// TIA Portal V15.1 export
// export: Created 2024-06-21T08:41:02.8317921Z, ExportSetting WithDefaults, DisplayName Totally Integrated Automation Portal, DisplayVersion V15.1 Update 5, DisplayName TIA Portal Openness, DisplayVersion V15.1 Update 5, DisplayName SINAMICS Startdrive Advanced, DisplayVersion V15.1, DisplayName G130, G150, S120, S150, SINAMICS MV, S210, DisplayVersion V15.1, DisplayName G110M, G120, G120C, G120D, G120P, DisplayVersion V15.1, DisplayName STEP 7 Professional, DisplayVersion V15.1 Update 5, DisplayName STEP 7 Safety, DisplayVersion V15.1, DisplayName WinCC Professional, DisplayVersion V15.1 Update 5, DisplayName SIMATIC Visualization Architect, DisplayVersion V15.1
FUNCTION_BLOCK "LProcModeSelector"   // FB1708, FBD
TITLE = LModeSelector
{ S7_Optimized_Access := 'FALSE' }
AUTHOR : VCC
FAMILY : Control
NAME : ModeSel
VERSION : 1.0
// ================================================================================
// This module handles that only one mode is selected in the modezon, it also 
// handle interlocking between the HMIs. Each modezone can have 5 HMI.
// ================================================================================
// stored: AutoNumber false, IsIECCheckEnabled false, SetENOAutomatically False, UDAEnableTagReadback false
   VAR_INPUT
      I_StartPB { ExternalAccessible := 'False'; ExternalVisible := 'False'; ExternalWritable := 'False'} : Bool;   // Summary of Start buttons
      I_AlarmResetPB { ExternalAccessible := 'False'; ExternalVisible := 'False'; ExternalWritable := 'False'} : Bool;   // Summary of Alarm reset buttons
      I_SafetyNotOk { ExternalAccessible := 'False'; ExternalVisible := 'False'; ExternalWritable := 'False'} : Bool;   // Safety is not ok
      I_FailSafeResetAck { ExternalAccessible := 'False'; ExternalVisible := 'False'; ExternalWritable := 'False'} : Bool;   // F_Ack_Op FB in safety program is requesting value 9 on FailSafeReset output
      I_FailSafeAckID { ExternalAccessible := 'False'; ExternalVisible := 'False'; ExternalWritable := 'False'} : Int;   // F_Ack ID
      I_HMI1ForceMan { ExternalAccessible := 'False'; ExternalVisible := 'False'; ExternalWritable := 'False'} : Bool;   // Forced manual selected on HMI1
      I_HMI1SetPB { ExternalAccessible := 'False'; ExternalVisible := 'False'; ExternalWritable := 'False'} : Bool;   // Set PB activated on HMI1
      I_HMI1ResetPB { ExternalAccessible := 'False'; ExternalVisible := 'False'; ExternalWritable := 'False'} : Bool;   // Reset PB activated on HMI1
      I_HMI1StartPB { ExternalAccessible := 'False'; ExternalVisible := 'False'; ExternalWritable := 'False'} : Bool;   // Start PB activated on HMI1
      I_HMI1AlarmResetPB { ExternalAccessible := 'False'; ExternalVisible := 'False'; ExternalWritable := 'False'} : Bool;   // AlarmReset PB activated on HMI1
      I_HMI2ForceMan { ExternalAccessible := 'False'; ExternalVisible := 'False'; ExternalWritable := 'False'} : Bool;   // Forced manual selected on HMI2
      I_HMI2SetPB { ExternalAccessible := 'False'; ExternalVisible := 'False'; ExternalWritable := 'False'} : Bool;   // Set PB activated on HMI2
      I_HMI2ResetPB { ExternalAccessible := 'False'; ExternalVisible := 'False'; ExternalWritable := 'False'} : Bool;   // Reset PB activated on HMI2
      I_HMI2StartPB { ExternalAccessible := 'False'; ExternalVisible := 'False'; ExternalWritable := 'False'} : Bool;   // Start PB activated on HMI2
      I_HMI2AlarmResetPB { ExternalAccessible := 'False'; ExternalVisible := 'False'; ExternalWritable := 'False'} : Bool;   // AlarmReset PB activated on HMI2
      I_HMI3ForceMan { ExternalAccessible := 'False'; ExternalVisible := 'False'; ExternalWritable := 'False'} : Bool;   // Forced manual selected on HMI3
      I_HMI3SetPB { ExternalAccessible := 'False'; ExternalVisible := 'False'; ExternalWritable := 'False'} : Bool;   // Set PB activated on HMI3
      I_HMI3ResetPB { ExternalAccessible := 'False'; ExternalVisible := 'False'; ExternalWritable := 'False'} : Bool;   // Reset PB activated on HMI3
      I_HMI3StartPB { ExternalAccessible := 'False'; ExternalVisible := 'False'; ExternalWritable := 'False'} : Bool;   // Start PB activated on HMI
      I_HMI3AlarmResetPB { ExternalAccessible := 'False'; ExternalVisible := 'False'; ExternalWritable := 'False'} : Bool;   // AlarmReset PB activated on HMI3
      I_HMI4ForceMan { ExternalAccessible := 'False'; ExternalVisible := 'False'; ExternalWritable := 'False'} : Bool;   // Forced manual selected on HMI4
      I_HMI4SetPB { ExternalAccessible := 'False'; ExternalVisible := 'False'; ExternalWritable := 'False'} : Bool;   // Set PB activated on HMI4
      I_HMI4ResetPB { ExternalAccessible := 'False'; ExternalVisible := 'False'; ExternalWritable := 'False'} : Bool;   // Reset PB activated on HMI4
      I_HMI4StartPB { ExternalAccessible := 'False'; ExternalVisible := 'False'; ExternalWritable := 'False'} : Bool;   // Start PB activated on HMI4
      I_HMI4AlarmResetPB { ExternalAccessible := 'False'; ExternalVisible := 'False'; ExternalWritable := 'False'} : Bool;   // AlarmReset PB activated on HMI4
      I_HMI5ForceMan { ExternalAccessible := 'False'; ExternalVisible := 'False'; ExternalWritable := 'False'} : Bool;   // Forced manual selected on HMI5
      I_HMI5SetPB { ExternalAccessible := 'False'; ExternalVisible := 'False'; ExternalWritable := 'False'} : Bool;   // Set PB activated on HMI5
      I_HMI5ResetPB { ExternalAccessible := 'False'; ExternalVisible := 'False'; ExternalWritable := 'False'} : Bool;   // Reset PB activated on HMI5
      I_HMI5StartPB { ExternalAccessible := 'False'; ExternalVisible := 'False'; ExternalWritable := 'False'} : Bool;   // Start PB activated on HMI5
      I_HMI5AlarmResetPB { ExternalAccessible := 'False'; ExternalVisible := 'False'; ExternalWritable := 'False'} : Bool;   // AlarmReset PB activated on HMI5
   END_VAR
   VAR_OUTPUT
      O_PBSetPBResetAllAutoSel { ExternalAccessible := 'False'; ExternalVisible := 'False'; ExternalWritable := 'False'} : Struct   // Set PB activated - Reset PB activated - All HMI Auto selected
         HMI1SetPB { ExternalAccessible := 'False'; ExternalVisible := 'False'; ExternalWritable := 'False'} : Bool;   // Set PB activated on HMI1
         HMI1ResetPB { ExternalAccessible := 'False'; ExternalVisible := 'False'; ExternalWritable := 'False'} : Bool;   // Reset PB activated on HMI1
         HMI1AllHMIAutoSel { ExternalAccessible := 'False'; ExternalVisible := 'False'; ExternalWritable := 'False'} : Bool;   // All HMI Auto selected on HMI1
         HMI2SetPB { ExternalAccessible := 'False'; ExternalVisible := 'False'; ExternalWritable := 'False'} : Bool;   // Set PB activated on HMI2
         HMI2ResetPB { ExternalAccessible := 'False'; ExternalVisible := 'False'; ExternalWritable := 'False'} : Bool;   // Reset PB activated on HMI2
         HMI2AllHMIAutoSel { ExternalAccessible := 'False'; ExternalVisible := 'False'; ExternalWritable := 'False'} : Bool;   // All HMI Auto selected on HMI2
         HMI3SetPB { ExternalAccessible := 'False'; ExternalVisible := 'False'; ExternalWritable := 'False'} : Bool;   // Set PB activated on HMI3
         HMI3ResetPB { ExternalAccessible := 'False'; ExternalVisible := 'False'; ExternalWritable := 'False'} : Bool;   // Reset PB activated on HMI3
         HMI3AllHMIAutoSel { ExternalAccessible := 'False'; ExternalVisible := 'False'; ExternalWritable := 'False'} : Bool;   // All HMI Auto selected on HMI3
         HMI4SetPB { ExternalAccessible := 'False'; ExternalVisible := 'False'; ExternalWritable := 'False'} : Bool;   // Set PB activated on HMI4
         HMI4ResetPB { ExternalAccessible := 'False'; ExternalVisible := 'False'; ExternalWritable := 'False'} : Bool;   // Reset PB activated on HMI4
         HMI4AllHMIAutoSel { ExternalAccessible := 'False'; ExternalVisible := 'False'; ExternalWritable := 'False'} : Bool;   // All HMI Auto selected on HMI4
         HMI5SetPB { ExternalAccessible := 'False'; ExternalVisible := 'False'; ExternalWritable := 'False'} : Bool;   // Set PB activated on HMI5
         HMI5ResetPB { ExternalAccessible := 'False'; ExternalVisible := 'False'; ExternalWritable := 'False'} : Bool;   // Reset PB activated on HMI5
         HMI5AllHMIAutoSel { ExternalAccessible := 'False'; ExternalVisible := 'False'; ExternalWritable := 'False'} : Bool;   // All HMI Auto selected on HMI5
         StartPBSel { ExternalAccessible := 'False'; ExternalVisible := 'False'; ExternalWritable := 'False'} : Bool;   // Start is activated
         AlarmResetPBSel { ExternalAccessible := 'False'; ExternalVisible := 'False'; ExternalWritable := 'False'} : Bool;   // Alarm reset is activated
      END_STRUCT;
   END_VAR
   VAR_IN_OUT
      IO_FailsafeReset { ExternalAccessible := 'False'; ExternalVisible := 'False'; ExternalWritable := 'False'} : Int;   // Number to Failsafe to reset safety
   END_VAR
   VAR DB_SPECIFIC
      H_HMIHomeRunModeCmd : Word;   // Homerun Mode commands from HMI
      H_Anim : Word;   // Animation for HMI
      H_ActiveHMI : Int;   // Active HMI
      H_NameActiveHMI : String[25];   // Name of the Active HMI
      H_LockManTime : Int;   // Lock manual time
      H_HMI1ModeCmd : Word;   // Mode commands from HMI1
      H_HMI2ModeCmd : Word;   // Mode commands from HMI2
      H_HMI3ModeCmd : Word;   // Mode commands from HMI3
      H_HMI4ModeCmd : Word;   // Mode commands from HMI4
      H_HMI5ModeCmd : Word;   // Mode commands from HMI5. For operator panels, no S7_m_c
      HMI1AutoSel { ExternalAccessible := 'False'; ExternalVisible := 'False'; ExternalWritable := 'False'} : Bool;   // Auto selected on HMI1
      HMI1StepSel { ExternalAccessible := 'False'; ExternalVisible := 'False'; ExternalWritable := 'False'} : Bool;   // Step selected on HMI1
      HMI1HomeRunSel { ExternalAccessible := 'False'; ExternalVisible := 'False'; ExternalWritable := 'False'} : Bool;   // Homerun selected on HMI1
      HMI1ManualSel { ExternalAccessible := 'False'; ExternalVisible := 'False'; ExternalWritable := 'False'} : Bool;   // Manual selected on HMI1
      HMI1LockManual { ExternalAccessible := 'False'; ExternalVisible := 'False'; ExternalWritable := 'False'} : Bool;   // Lock manual for HMI1
      HMI1AllHMIAutoSel { ExternalAccessible := 'False'; ExternalVisible := 'False'; ExternalWritable := 'False'} : Bool;   // All HMI Auto selected on HMI1
      HMI1Start { ExternalAccessible := 'False'; ExternalVisible := 'False'; ExternalWritable := 'False'} : Bool;   // Start on HMI1
      HMI1AlarmReset { ExternalAccessible := 'False'; ExternalVisible := 'False'; ExternalWritable := 'False'} : Bool;   // AlarmReset on HMI1
      HMI1ResetTM { ExternalAccessible := 'False'; ExternalVisible := 'False'; ExternalWritable := 'False'} : Bool;   // Reset transport memory from HMI1
      HMI1ResetSeq { ExternalAccessible := 'False'; ExternalVisible := 'False'; ExternalWritable := 'False'} : Bool;   // Reset sequence from HMI1
      HMI1CycleFinished { ExternalAccessible := 'False'; ExternalVisible := 'False'; ExternalWritable := 'False'} : Bool;   // Cycle Finished from HMI1
      HMI1AlarmResetAck { ExternalAccessible := 'False'; ExternalVisible := 'False'; ExternalWritable := 'False'} : Bool;   // Alarm Reset acknowledge from HMI1
      HMI2AutoSel { ExternalAccessible := 'False'; ExternalVisible := 'False'; ExternalWritable := 'False'} : Bool;   // Auto selected on HMI2
      HMI2StepSel { ExternalAccessible := 'False'; ExternalVisible := 'False'; ExternalWritable := 'False'} : Bool;   // Step selected on HMI2
      HMI2HomeRunSel { ExternalAccessible := 'False'; ExternalVisible := 'False'; ExternalWritable := 'False'} : Bool;   // Homerun selected on HMI2
      HMI2ManualSel { ExternalAccessible := 'False'; ExternalVisible := 'False'; ExternalWritable := 'False'} : Bool;   // Manual selected on HMI2
      HMI2LockManual { ExternalAccessible := 'False'; ExternalVisible := 'False'; ExternalWritable := 'False'} : Bool;   // Lock manual for HMI2
      HMI2AllHMIAutoSel { ExternalAccessible := 'False'; ExternalVisible := 'False'; ExternalWritable := 'False'} : Bool;   // All HMI Auto selected on HMI2
      HMI2Start { ExternalAccessible := 'False'; ExternalVisible := 'False'; ExternalWritable := 'False'} : Bool;   // Start on HMI2
      HMI2AlarmReset { ExternalAccessible := 'False'; ExternalVisible := 'False'; ExternalWritable := 'False'} : Bool;   // AlarmReset on HMI2
      HMI2ResetTM { ExternalAccessible := 'False'; ExternalVisible := 'False'; ExternalWritable := 'False'} : Bool;   // Reset transport memory from HMI2
      HMI2ResetSeq { ExternalAccessible := 'False'; ExternalVisible := 'False'; ExternalWritable := 'False'} : Bool;   // Reset sequence from HMI2
      HMI2CycleFinished { ExternalAccessible := 'False'; ExternalVisible := 'False'; ExternalWritable := 'False'} : Bool;   // Cycle Finished from HMI2
      HMI2AlarmResetAck { ExternalAccessible := 'False'; ExternalVisible := 'False'; ExternalWritable := 'False'} : Bool;   // Alarm Reset acknowledge from HMI2
      HMI3AutoSel { ExternalAccessible := 'False'; ExternalVisible := 'False'; ExternalWritable := 'False'} : Bool;   // Auto selected on HMI3
      HMI3StepSel { ExternalAccessible := 'False'; ExternalVisible := 'False'; ExternalWritable := 'False'} : Bool;   // Step selected on HMI3
      HMI3HomeRunSel { ExternalAccessible := 'False'; ExternalVisible := 'False'; ExternalWritable := 'False'} : Bool;   // Homerun selected on HMI3
      HMI3ManualSel { ExternalAccessible := 'False'; ExternalVisible := 'False'; ExternalWritable := 'False'} : Bool;   // Manual selected on HMI3
      HMI3LockManual { ExternalAccessible := 'False'; ExternalVisible := 'False'; ExternalWritable := 'False'} : Bool;   // Lock manual for HMI3
      HMI3AllHMIAutoSel { ExternalAccessible := 'False'; ExternalVisible := 'False'; ExternalWritable := 'False'} : Bool;   // All HMI Auto selected on HMI3
      HMI3Start { ExternalAccessible := 'False'; ExternalVisible := 'False'; ExternalWritable := 'False'} : Bool;   // Start on HMI3
      HMI3AlarmReset { ExternalAccessible := 'False'; ExternalVisible := 'False'; ExternalWritable := 'False'} : Bool;   // AlarmReset on HMI3
      HMI3ResetTM { ExternalAccessible := 'False'; ExternalVisible := 'False'; ExternalWritable := 'False'} : Bool;   // Reset transport memory from HMI3
      HMI3ResetSeq { ExternalAccessible := 'False'; ExternalVisible := 'False'; ExternalWritable := 'False'} : Bool;   // Reset sequence from HMI3
      HMI3CycleFinished { ExternalAccessible := 'False'; ExternalVisible := 'False'; ExternalWritable := 'False'} : Bool;   // Cycle Finished from HMI3
      HMI3AlarmResetAck { ExternalAccessible := 'False'; ExternalVisible := 'False'; ExternalWritable := 'False'} : Bool;   // Alarm Reset acknowledge from 3
      HMI4AutoSel { ExternalAccessible := 'False'; ExternalVisible := 'False'; ExternalWritable := 'False'} : Bool;   // Auto selected on HMI4
      HMI4StepSel { ExternalAccessible := 'False'; ExternalVisible := 'False'; ExternalWritable := 'False'} : Bool;   // Step selected on HMI4
      HMI4HomeRunSel { ExternalAccessible := 'False'; ExternalVisible := 'False'; ExternalWritable := 'False'} : Bool;   // Homerun selected on HMI4
      HMI4ManualSel { ExternalAccessible := 'False'; ExternalVisible := 'False'; ExternalWritable := 'False'} : Bool;   // Manual selected on HMI4
      HMI4LockManual { ExternalAccessible := 'False'; ExternalVisible := 'False'; ExternalWritable := 'False'} : Bool;   // Lock manual for HMI4
      HMI4AllHMIAutoSel { ExternalAccessible := 'False'; ExternalVisible := 'False'; ExternalWritable := 'False'} : Bool;   // All HMI Auto selected on HMI4
      HMI4Start { ExternalAccessible := 'False'; ExternalVisible := 'False'; ExternalWritable := 'False'} : Bool;   // Start on HMI4
      HMI4AlarmReset { ExternalAccessible := 'False'; ExternalVisible := 'False'; ExternalWritable := 'False'} : Bool;   // AlarmReset on HMI4
      HMI4ResetTM { ExternalAccessible := 'False'; ExternalVisible := 'False'; ExternalWritable := 'False'} : Bool;   // Reset transport memory from HMI4
      HMI4ResetSeq { ExternalAccessible := 'False'; ExternalVisible := 'False'; ExternalWritable := 'False'} : Bool;   // Reset sequence from HMI4
      HMI4CycleFinished { ExternalAccessible := 'False'; ExternalVisible := 'False'; ExternalWritable := 'False'} : Bool;   // Cycle Finished from HMI4
      HMI4AlarmResetAck { ExternalAccessible := 'False'; ExternalVisible := 'False'; ExternalWritable := 'False'} : Bool;   // Alarm Reset acknowledge from HMI4
      HMI5AutoSel { ExternalAccessible := 'False'; ExternalVisible := 'False'; ExternalWritable := 'False'} : Bool;   // Auto selected on HMI5
      HMI5StepSel { ExternalAccessible := 'False'; ExternalVisible := 'False'; ExternalWritable := 'False'} : Bool;   // Step selected on HMI5
      HMI5HomeRunSel { ExternalAccessible := 'False'; ExternalVisible := 'False'; ExternalWritable := 'False'} : Bool;   // Homerun selected on HMI5
      HMI5ManualSel { ExternalAccessible := 'False'; ExternalVisible := 'False'; ExternalWritable := 'False'} : Bool;   // Manual selected on HMI5
      HMI5LockManual { ExternalAccessible := 'False'; ExternalVisible := 'False'; ExternalWritable := 'False'} : Bool;   // Lock manual for HMI5
      HMI5AllHMIAutoSel { ExternalAccessible := 'False'; ExternalVisible := 'False'; ExternalWritable := 'False'} : Bool;   // All HMI Auto selected on HMI5
      HMI5Start { ExternalAccessible := 'False'; ExternalVisible := 'False'; ExternalWritable := 'False'} : Bool;   // Start on HMI5
      HMI5AlarmReset { ExternalAccessible := 'False'; ExternalVisible := 'False'; ExternalWritable := 'False'} : Bool;   // AlarmReset on HMI5
      HMI5ResetTM { ExternalAccessible := 'False'; ExternalVisible := 'False'; ExternalWritable := 'False'} : Bool;   // Reset transport memory from HMI5
      HMI5ResetSeq { ExternalAccessible := 'False'; ExternalVisible := 'False'; ExternalWritable := 'False'} : Bool;   // Reset sequence from HMI5
      HMI5CycleFinished { ExternalAccessible := 'False'; ExternalVisible := 'False'; ExternalWritable := 'False'} : Bool;   // Cycle Finished from HMI5
      HMI5AlarmResetAck { ExternalAccessible := 'False'; ExternalVisible := 'False'; ExternalWritable := 'False'} : Bool;   // Alarm Reset acknowledge from HMI5
      HMIHomeRunRedo { ExternalAccessible := 'False'; ExternalVisible := 'False'; ExternalWritable := 'False'} : Bool;   // Redo after homerun from HMI
      HMIHomeRunWorkDone { ExternalAccessible := 'False'; ExternalVisible := 'False'; ExternalWritable := 'False'} : Bool;   // WorkDone after homerun from HMI
      LockManualTimeout { ExternalAccessible := 'False'; ExternalVisible := 'False'; ExternalWritable := 'False'} : Bool;   // Lock manual button timeout
      AllHmiAutoSel { ExternalAccessible := 'False'; ExternalVisible := 'False'; ExternalWritable := 'False'} : Bool;   // All Hmi Auto selected
      AlarmResetPBSel { ExternalAccessible := 'False'; ExternalVisible := 'False'; ExternalWritable := 'False'} : Bool;   // Alarm reset is activated
      AlarmResetPBSelReset { ExternalAccessible := 'False'; ExternalVisible := 'False'; ExternalWritable := 'False'} : Bool;   // Reset AlarmResetPBSel after predefined time
      AlarmResetPBSelResetPE { ExternalAccessible := 'False'; ExternalVisible := 'False'; ExternalWritable := 'False'} : Bool;   // Positive edge of AlarmResetPbSelReset
      FailSafeReset6Pulse { ExternalAccessible := 'False'; ExternalVisible := 'False'; ExternalWritable := 'False'} : Bool;   // Pulse to set value 6 on FailSafeReset Output
      FailSafeReset9Pulse { ExternalAccessible := 'False'; ExternalVisible := 'False'; ExternalWritable := 'False'} : Bool;   // Pulse to set value 9 on FailSafeReset Output
      ResetAlarmAckMemPulse { ExternalAccessible := 'False'; ExternalVisible := 'False'; ExternalWritable := 'False'} : Bool;   // Pulse to reset AlarmResetAckMem on negative edge of I_FailSafeResetAck
      AlarmResetAckMem { ExternalAccessible := 'False'; ExternalVisible := 'False'; ExternalWritable := 'False'} : Bool;   // memory : Pushbutton AlarmResetAck has been pushed on HMI
      StartPBSel { ExternalAccessible := 'False'; ExternalVisible := 'False'; ExternalWritable := 'False'} : Bool;   // Summary of the Start push buttons
      HMIStartPE { ExternalAccessible := 'False'; ExternalVisible := 'False'; ExternalWritable := 'False'} : Bool;   // Positive edge on start button from HMI
      HMIResetTMPE { ExternalAccessible := 'False'; ExternalVisible := 'False'; ExternalWritable := 'False'} : Bool;   // Positive edge on ResetTM button from HMI
      HMIResetSeqPE { ExternalAccessible := 'False'; ExternalVisible := 'False'; ExternalWritable := 'False'} : Bool;   // Positive edge on ResetSeq button from HMI
      HMIAlarmResetAckPE { ExternalAccessible := 'False'; ExternalVisible := 'False'; ExternalWritable := 'False'} : Bool;   // Positive edge on AlarmResetAck button from HMI
      HMILockManualPE { ExternalAccessible := 'False'; ExternalVisible := 'False'; ExternalWritable := 'False'} : Bool;   // Positive edge on LockManual button from HMI
      FailsafeReset { ExternalAccessible := 'False'; ExternalVisible := 'False'; ExternalWritable := 'False'} : Int;   // Number to Failsafe to reset safety
      ActiveHMI { ExternalAccessible := 'False'; ExternalVisible := 'False'; ExternalWritable := 'False'} : Int;   // Help memory for Active HMI
   END_VAR
   VAR
      TimerLockMan { ExternalAccessible := 'False'; ExternalVisible := 'False'; ExternalWritable := 'False'; S7_SetPoint := 'True'} : "LTimer";   // Timer on Lock manual
      TimerAlarmResetPB { ExternalAccessible := 'False'; ExternalVisible := 'False'; ExternalWritable := 'False'; S7_SetPoint := 'True'} : "LTimer";   // Timer on alarm reset
   END_VAR
   VAR_TEMP
      PHMI1AutoSel : Bool;   // Pulse Auto selected HMI1
      PHMI2AutoSel : Bool;   // Pulse Auto selected HMI2
      PHMI3AutoSel : Bool;   // Pulse Auto selected HMI3
      PHMI4AutoSel : Bool;   // Pulse Auto selected HMI4
      PHMI5AutoSel : Bool;   // Pulse Auto selected HMI5
   END_VAR
   VAR_TEMP   // added for the SCL form of the ladder/FBD networks
      _w1 : Bool;
      _w2 : Bool;
      _w3 : Bool;
      _w4 : Bool;
      _w5 : Bool;
   END_VAR
BEGIN

REGION Network 1: **** 1 - Inputs **** Extract the modeselection from HMI 1
   // Extract the modeselection from HMI 1
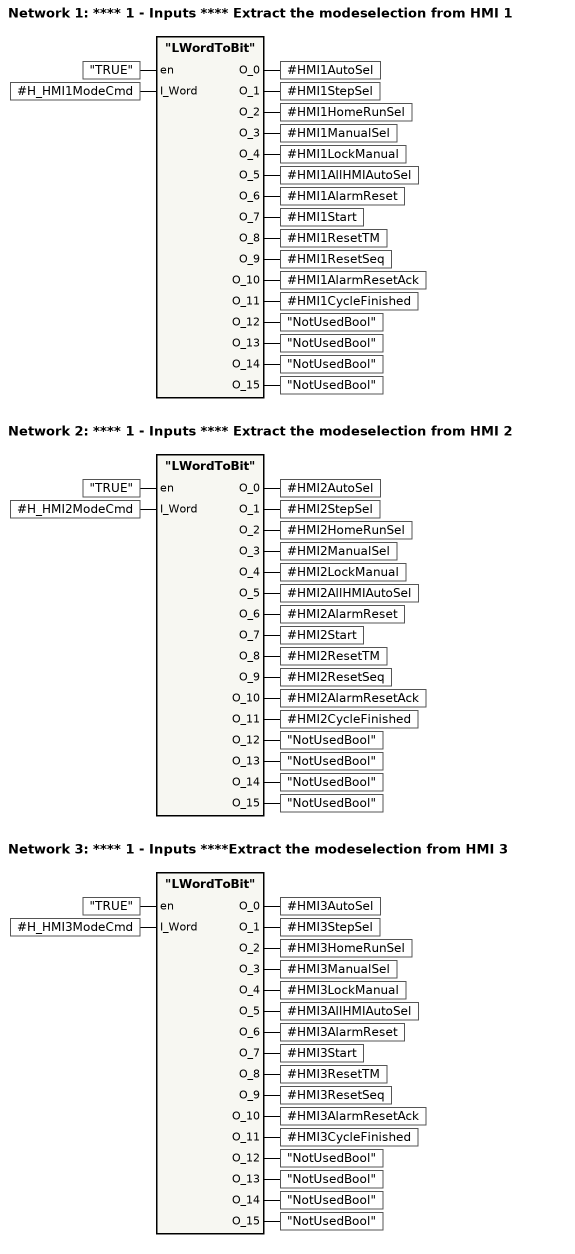
   IF "TRUE" THEN
       "LWordToBit"(I_Word := #H_HMI1ModeCmd,
                    O_0 => #HMI1AutoSel,
                    O_1 => #HMI1StepSel,
                    O_2 => #HMI1HomeRunSel,
                    O_3 => #HMI1ManualSel,
                    O_4 => #HMI1LockManual,
                    O_5 => #HMI1AllHMIAutoSel,
                    O_6 => #HMI1AlarmReset,
                    O_7 => #HMI1Start,
                    O_8 => #HMI1ResetTM,
                    O_9 => #HMI1ResetSeq,
                    O_10 => #HMI1AlarmResetAck,
                    O_11 => #HMI1CycleFinished,
                    O_12 => "NotUsedBool",
                    O_13 => "NotUsedBool",
                    O_14 => "NotUsedBool",
                    O_15 => "NotUsedBool");
   END_IF;
END_REGION

REGION Network 2: **** 1 - Inputs **** Extract the modeselection from HMI 2
   // Extract the modeselection from HMI 2
   IF "TRUE" THEN
       "LWordToBit"(I_Word := #H_HMI2ModeCmd,
                    O_0 => #HMI2AutoSel,
                    O_1 => #HMI2StepSel,
                    O_2 => #HMI2HomeRunSel,
                    O_3 => #HMI2ManualSel,
                    O_4 => #HMI2LockManual,
                    O_5 => #HMI2AllHMIAutoSel,
                    O_6 => #HMI2AlarmReset,
                    O_7 => #HMI2Start,
                    O_8 => #HMI2ResetTM,
                    O_9 => #HMI2ResetSeq,
                    O_10 => #HMI2AlarmResetAck,
                    O_11 => #HMI2CycleFinished,
                    O_12 => "NotUsedBool",
                    O_13 => "NotUsedBool",
                    O_14 => "NotUsedBool",
                    O_15 => "NotUsedBool");
   END_IF;
END_REGION

REGION Network 3: **** 1 - Inputs ****Extract the modeselection from HMI 3
   // Extract the modeselection from HMI 3
   IF "TRUE" THEN
       "LWordToBit"(I_Word := #H_HMI3ModeCmd,
                    O_0 => #HMI3AutoSel,
                    O_1 => #HMI3StepSel,
                    O_2 => #HMI3HomeRunSel,
                    O_3 => #HMI3ManualSel,
                    O_4 => #HMI3LockManual,
                    O_5 => #HMI3AllHMIAutoSel,
                    O_6 => #HMI3AlarmReset,
                    O_7 => #HMI3Start,
                    O_8 => #HMI3ResetTM,
                    O_9 => #HMI3ResetSeq,
                    O_10 => #HMI3AlarmResetAck,
                    O_11 => #HMI3CycleFinished,
                    O_12 => "NotUsedBool",
                    O_13 => "NotUsedBool",
                    O_14 => "NotUsedBool",
                    O_15 => "NotUsedBool");
   END_IF;
END_REGION

REGION Network 4: **** 1 - Inputs **** Extract the modeselection from HMI 4
   // Extract the modeselection from HMI 4
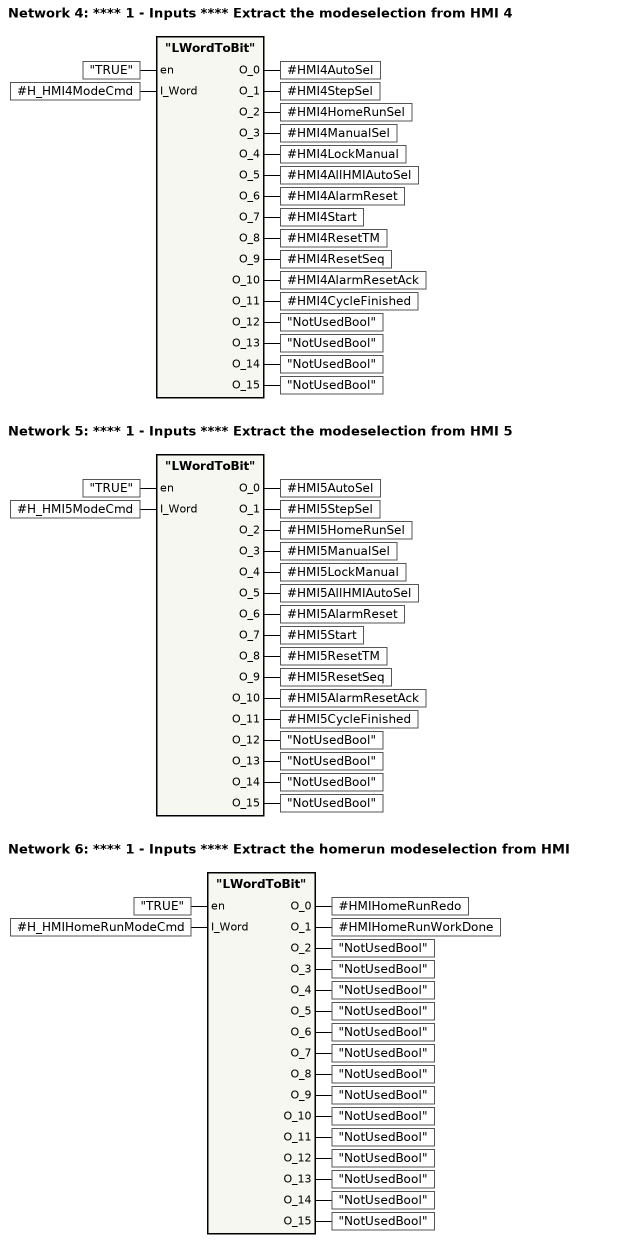
   IF "TRUE" THEN
       "LWordToBit"(I_Word := #H_HMI4ModeCmd,
                    O_0 => #HMI4AutoSel,
                    O_1 => #HMI4StepSel,
                    O_2 => #HMI4HomeRunSel,
                    O_3 => #HMI4ManualSel,
                    O_4 => #HMI4LockManual,
                    O_5 => #HMI4AllHMIAutoSel,
                    O_6 => #HMI4AlarmReset,
                    O_7 => #HMI4Start,
                    O_8 => #HMI4ResetTM,
                    O_9 => #HMI4ResetSeq,
                    O_10 => #HMI4AlarmResetAck,
                    O_11 => #HMI4CycleFinished,
                    O_12 => "NotUsedBool",
                    O_13 => "NotUsedBool",
                    O_14 => "NotUsedBool",
                    O_15 => "NotUsedBool");
   END_IF;
END_REGION

REGION Network 5: **** 1 - Inputs **** Extract the modeselection from HMI 5
   // Extract the modeselection from HMI 5
   IF "TRUE" THEN
       "LWordToBit"(I_Word := #H_HMI5ModeCmd,
                    O_0 => #HMI5AutoSel,
                    O_1 => #HMI5StepSel,
                    O_2 => #HMI5HomeRunSel,
                    O_3 => #HMI5ManualSel,
                    O_4 => #HMI5LockManual,
                    O_5 => #HMI5AllHMIAutoSel,
                    O_6 => #HMI5AlarmReset,
                    O_7 => #HMI5Start,
                    O_8 => #HMI5ResetTM,
                    O_9 => #HMI5ResetSeq,
                    O_10 => #HMI5AlarmResetAck,
                    O_11 => #HMI5CycleFinished,
                    O_12 => "NotUsedBool",
                    O_13 => "NotUsedBool",
                    O_14 => "NotUsedBool",
                    O_15 => "NotUsedBool");
   END_IF;
END_REGION

REGION Network 6: **** 1 - Inputs **** Extract the homerun modeselection from HMI
   // Extract the homerun modeselection from HMI
   IF "TRUE" THEN
       "LWordToBit"(I_Word := #H_HMIHomeRunModeCmd,
                    O_0 => #HMIHomeRunRedo,
                    O_1 => #HMIHomeRunWorkDone,
                    O_2 => "NotUsedBool",
                    O_3 => "NotUsedBool",
                    O_4 => "NotUsedBool",
                    O_5 => "NotUsedBool",
                    O_6 => "NotUsedBool",
                    O_7 => "NotUsedBool",
                    O_8 => "NotUsedBool",
                    O_9 => "NotUsedBool",
                    O_10 => "NotUsedBool",
                    O_11 => "NotUsedBool",
                    O_12 => "NotUsedBool",
                    O_13 => "NotUsedBool",
                    O_14 => "NotUsedBool",
                    O_15 => "NotUsedBool");
   END_IF;
END_REGION

REGION Network 7: **** 1 - Inputs **** All HMI Auto selected
   // All HMI Auto selected
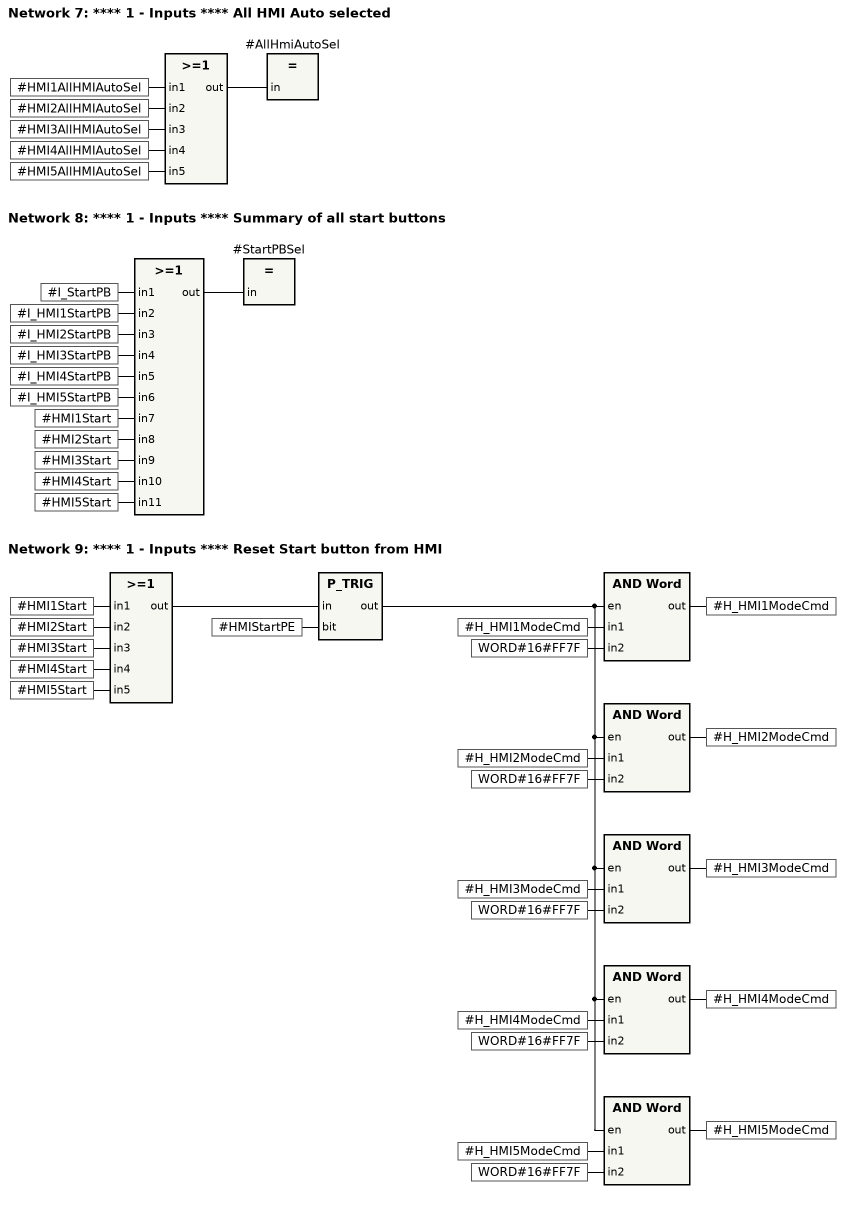
   #AllHmiAutoSel := #HMI1AllHMIAutoSel OR #HMI2AllHMIAutoSel OR #HMI3AllHMIAutoSel OR #HMI4AllHMIAutoSel OR #HMI5AllHMIAutoSel;
END_REGION

REGION Network 8: **** 1 - Inputs **** Summary of all start buttons
   // Summary of all start buttons
   #StartPBSel := #I_StartPB OR #I_HMI1StartPB OR #I_HMI2StartPB OR #I_HMI3StartPB OR #I_HMI4StartPB OR #I_HMI5StartPB OR #HMI1Start OR #HMI2Start OR #HMI3Start OR #HMI4Start OR #HMI5Start;
END_REGION

REGION Network 9: **** 1 - Inputs **** Reset Start button from HMI
   // Reset Start button from HMI
   #_w1 := #HMI1Start OR #HMI2Start OR #HMI3Start OR #HMI4Start OR #HMI5Start;
   #_w2 := #_w1 AND NOT #HMIStartPE;   // rising edge
   #HMIStartPE := #_w1;
   IF #_w2 THEN
       #H_HMI1ModeCmd := #H_HMI1ModeCmd AND WORD#16#FF7F;
       #H_HMI2ModeCmd := #H_HMI2ModeCmd AND WORD#16#FF7F;
       #H_HMI3ModeCmd := #H_HMI3ModeCmd AND WORD#16#FF7F;
       #H_HMI4ModeCmd := #H_HMI4ModeCmd AND WORD#16#FF7F;
       #H_HMI5ModeCmd := #H_HMI5ModeCmd AND WORD#16#FF7F;
   END_IF;
END_REGION

REGION Network 10: **** 1 - Inputs **** Summary of all alarm reset buttons
   // Summary of all alarm reset buttons
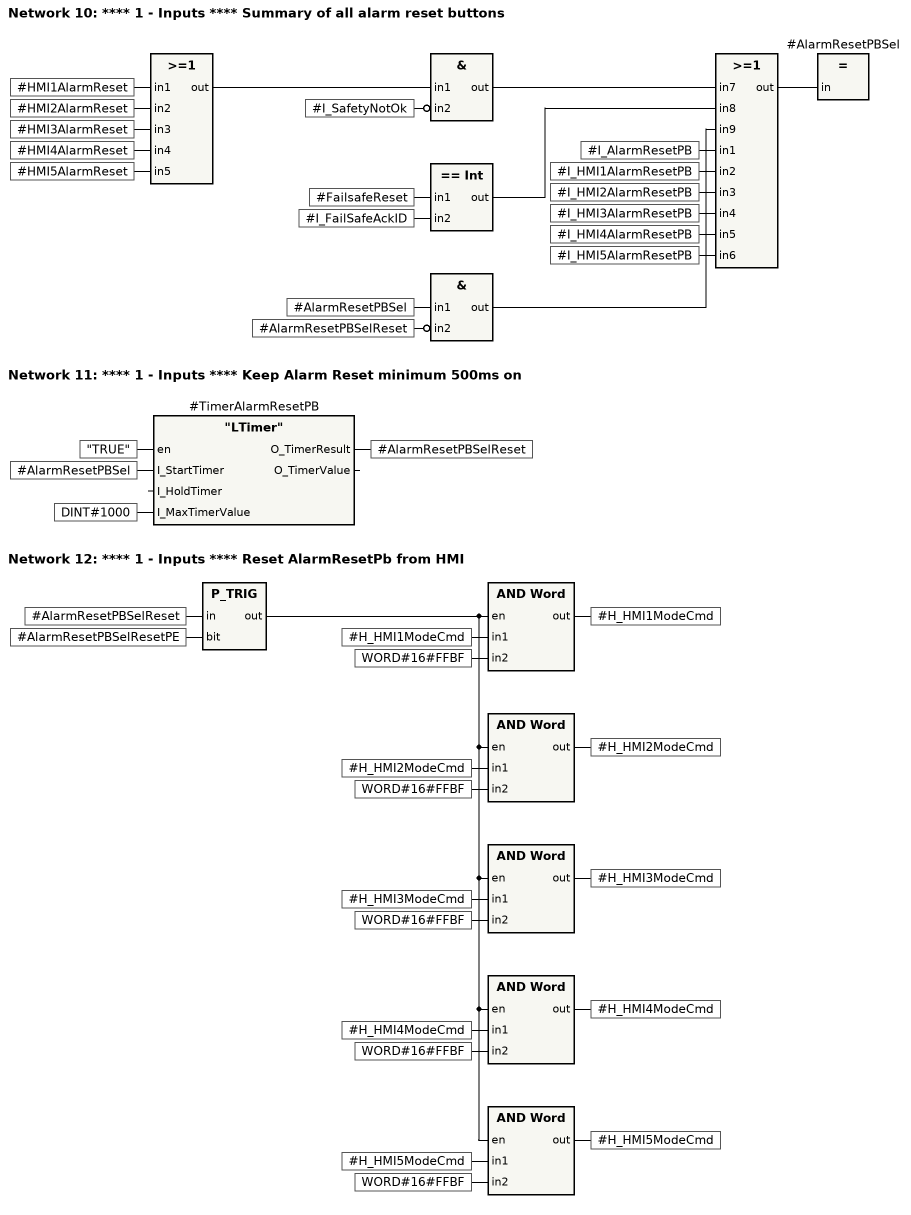
   #AlarmResetPBSel := ((#HMI1AlarmReset OR #HMI2AlarmReset OR #HMI3AlarmReset OR #HMI4AlarmReset OR #HMI5AlarmReset) AND NOT #I_SafetyNotOk) OR (#FailsafeReset = #I_FailSafeAckID) OR (#AlarmResetPBSel AND NOT #AlarmResetPBSelReset) OR #I_AlarmResetPB OR #I_HMI1AlarmResetPB OR #I_HMI2AlarmResetPB OR #I_HMI3AlarmResetPB OR #I_HMI4AlarmResetPB OR #I_HMI5AlarmResetPB;
END_REGION

REGION Network 11: **** 1 - Inputs **** Keep Alarm Reset minimum 500ms on
   // Keep Alarm Reset minimum 500ms on
   IF "TRUE" THEN
       #TimerAlarmResetPB(I_StartTimer := #AlarmResetPBSel,   // "LTimer"
                          I_MaxTimerValue := DINT#1000,
                          O_TimerResult => #AlarmResetPBSelReset);
   END_IF;
END_REGION

REGION Network 12: **** 1 - Inputs **** Reset AlarmResetPb from HMI
   // Reset AlarmResetPb from HMI
   #_w1 := #AlarmResetPBSelReset AND NOT #AlarmResetPBSelResetPE;   // rising edge
   #AlarmResetPBSelResetPE := #AlarmResetPBSelReset;
   IF #_w1 THEN
       #H_HMI1ModeCmd := #H_HMI1ModeCmd AND WORD#16#FFBF;
       #H_HMI2ModeCmd := #H_HMI2ModeCmd AND WORD#16#FFBF;
       #H_HMI3ModeCmd := #H_HMI3ModeCmd AND WORD#16#FFBF;
       #H_HMI4ModeCmd := #H_HMI4ModeCmd AND WORD#16#FFBF;
       #H_HMI5ModeCmd := #H_HMI5ModeCmd AND WORD#16#FFBF;
   END_IF;
END_REGION

REGION Network 13: **** 1 - Inputs **** Reset AlarmResetAckPb from HMI
   // Reset AlarmResetAckPb from HMI
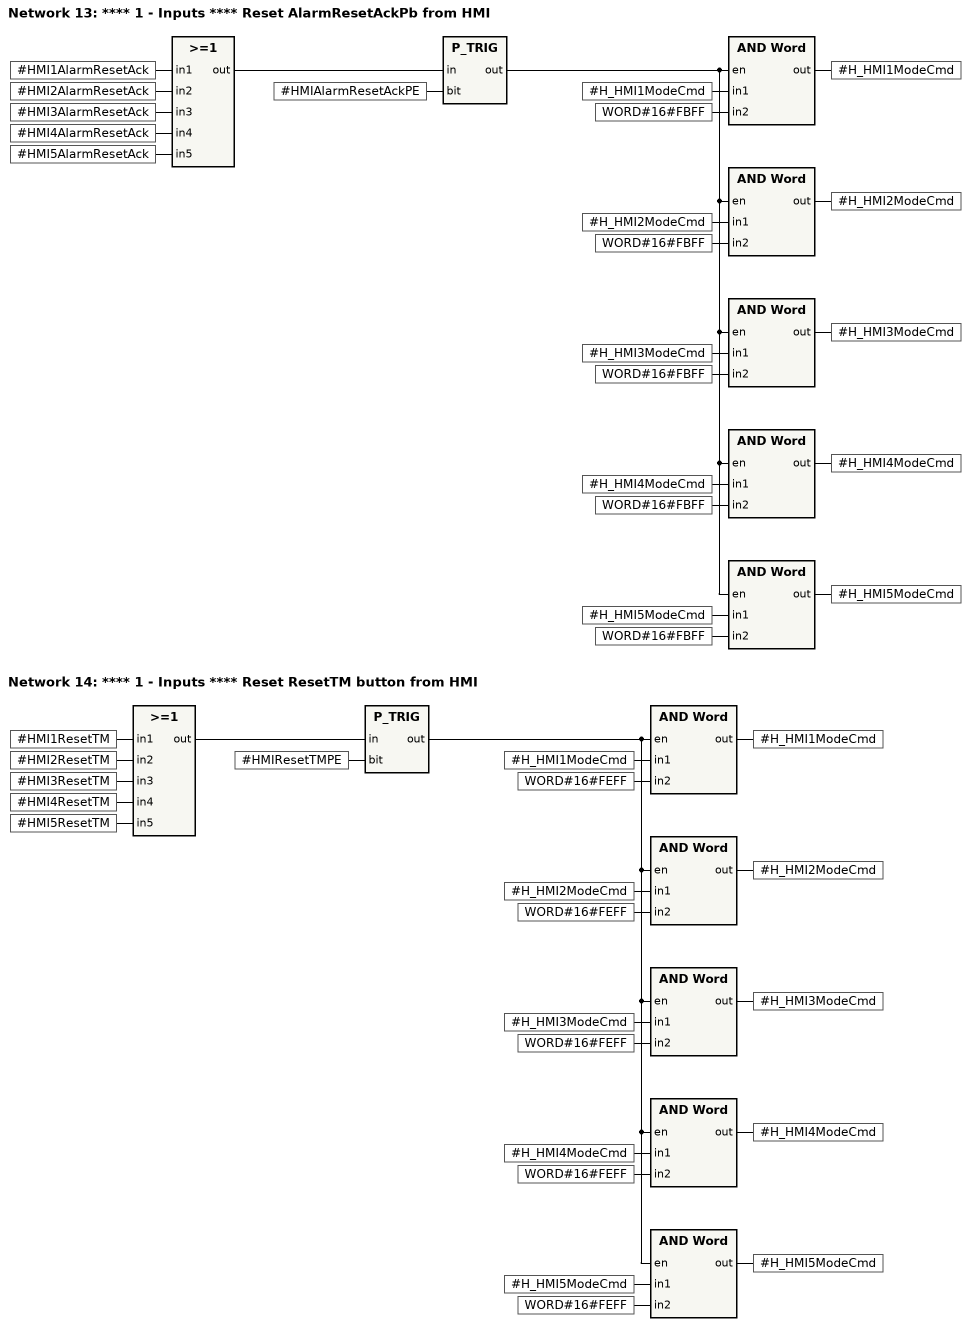
   #_w1 := #HMI1AlarmResetAck OR #HMI2AlarmResetAck OR #HMI3AlarmResetAck OR #HMI4AlarmResetAck OR #HMI5AlarmResetAck;
   #_w2 := #_w1 AND NOT #HMIAlarmResetAckPE;   // rising edge
   #HMIAlarmResetAckPE := #_w1;
   IF #_w2 THEN
       #H_HMI1ModeCmd := #H_HMI1ModeCmd AND WORD#16#FBFF;
       #H_HMI2ModeCmd := #H_HMI2ModeCmd AND WORD#16#FBFF;
       #H_HMI3ModeCmd := #H_HMI3ModeCmd AND WORD#16#FBFF;
       #H_HMI4ModeCmd := #H_HMI4ModeCmd AND WORD#16#FBFF;
       #H_HMI5ModeCmd := #H_HMI5ModeCmd AND WORD#16#FBFF;
   END_IF;
END_REGION

REGION Network 14: **** 1 - Inputs **** Reset ResetTM button from HMI
   // Reset ResetTM button from HMI
   #_w1 := #HMI1ResetTM OR #HMI2ResetTM OR #HMI3ResetTM OR #HMI4ResetTM OR #HMI5ResetTM;
   #_w2 := #_w1 AND NOT #HMIResetTMPE;   // rising edge
   #HMIResetTMPE := #_w1;
   IF #_w2 THEN
       #H_HMI1ModeCmd := #H_HMI1ModeCmd AND WORD#16#FEFF;
       #H_HMI2ModeCmd := #H_HMI2ModeCmd AND WORD#16#FEFF;
       #H_HMI3ModeCmd := #H_HMI3ModeCmd AND WORD#16#FEFF;
       #H_HMI4ModeCmd := #H_HMI4ModeCmd AND WORD#16#FEFF;
       #H_HMI5ModeCmd := #H_HMI5ModeCmd AND WORD#16#FEFF;
   END_IF;
END_REGION

REGION Network 15: **** 1 - Inputs **** Reset ResetSeq button from HMI
   // Reset ResetSeq button from HMI
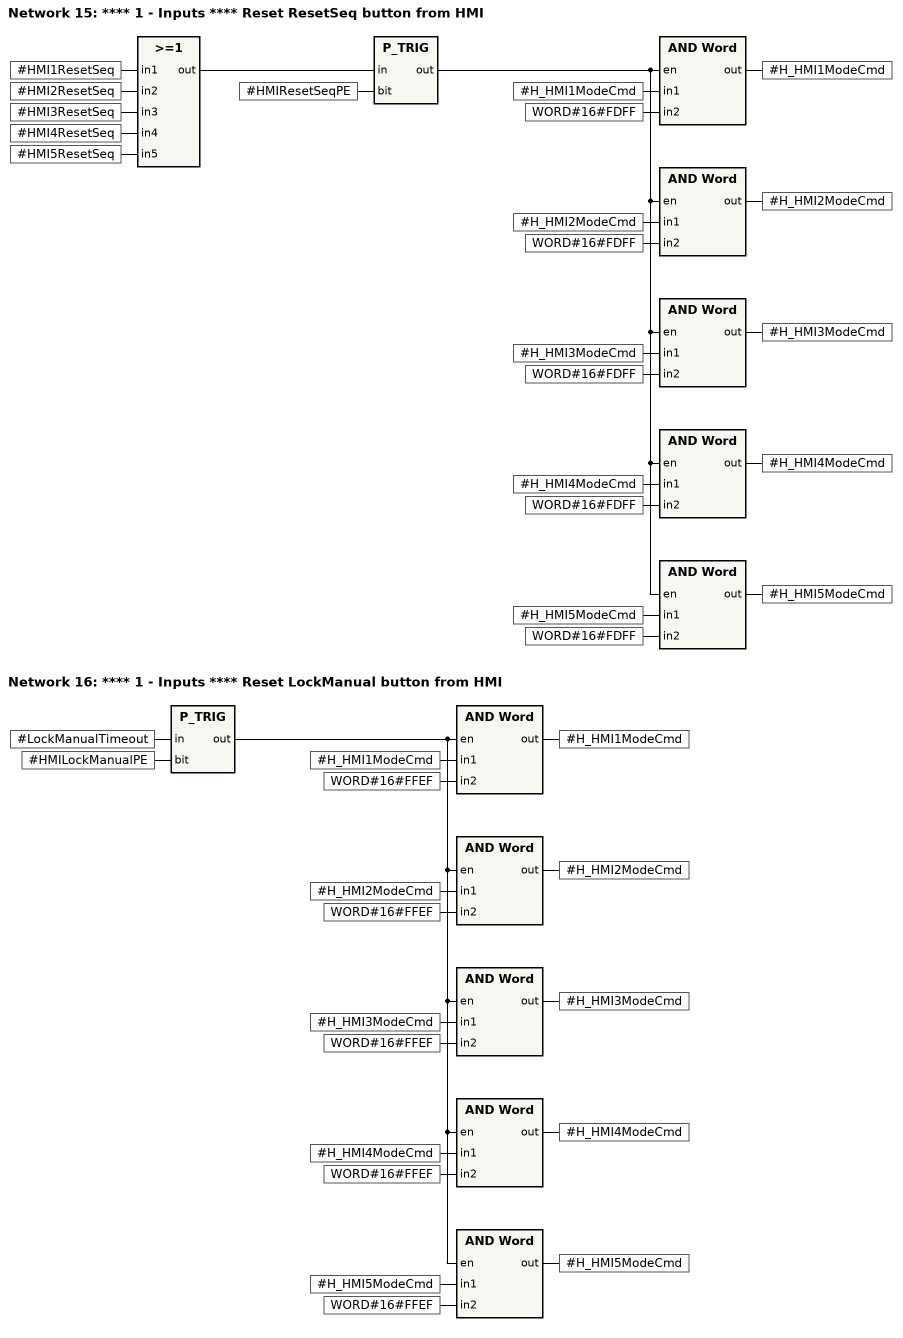
   #_w1 := #HMI1ResetSeq OR #HMI2ResetSeq OR #HMI3ResetSeq OR #HMI4ResetSeq OR #HMI5ResetSeq;
   #_w2 := #_w1 AND NOT #HMIResetSeqPE;   // rising edge
   #HMIResetSeqPE := #_w1;
   IF #_w2 THEN
       #H_HMI1ModeCmd := #H_HMI1ModeCmd AND WORD#16#FDFF;
       #H_HMI2ModeCmd := #H_HMI2ModeCmd AND WORD#16#FDFF;
       #H_HMI3ModeCmd := #H_HMI3ModeCmd AND WORD#16#FDFF;
       #H_HMI4ModeCmd := #H_HMI4ModeCmd AND WORD#16#FDFF;
       #H_HMI5ModeCmd := #H_HMI5ModeCmd AND WORD#16#FDFF;
   END_IF;
END_REGION

REGION Network 16: **** 1 - Inputs **** Reset LockManual button from HMI
   // Reset LockManual button from HMI
   #_w1 := #LockManualTimeout AND NOT #HMILockManualPE;   // rising edge
   #HMILockManualPE := #LockManualTimeout;
   IF #_w1 THEN
       #H_HMI1ModeCmd := #H_HMI1ModeCmd AND WORD#16#FFEF;
       #H_HMI2ModeCmd := #H_HMI2ModeCmd AND WORD#16#FFEF;
       #H_HMI3ModeCmd := #H_HMI3ModeCmd AND WORD#16#FFEF;
       #H_HMI4ModeCmd := #H_HMI4ModeCmd AND WORD#16#FFEF;
       #H_HMI5ModeCmd := #H_HMI5ModeCmd AND WORD#16#FFEF;
   END_IF;
END_REGION

REGION Network 17: **** 4.5 - Machine Status - Modes **** Reset activ HMI
   // Reset activ HMI
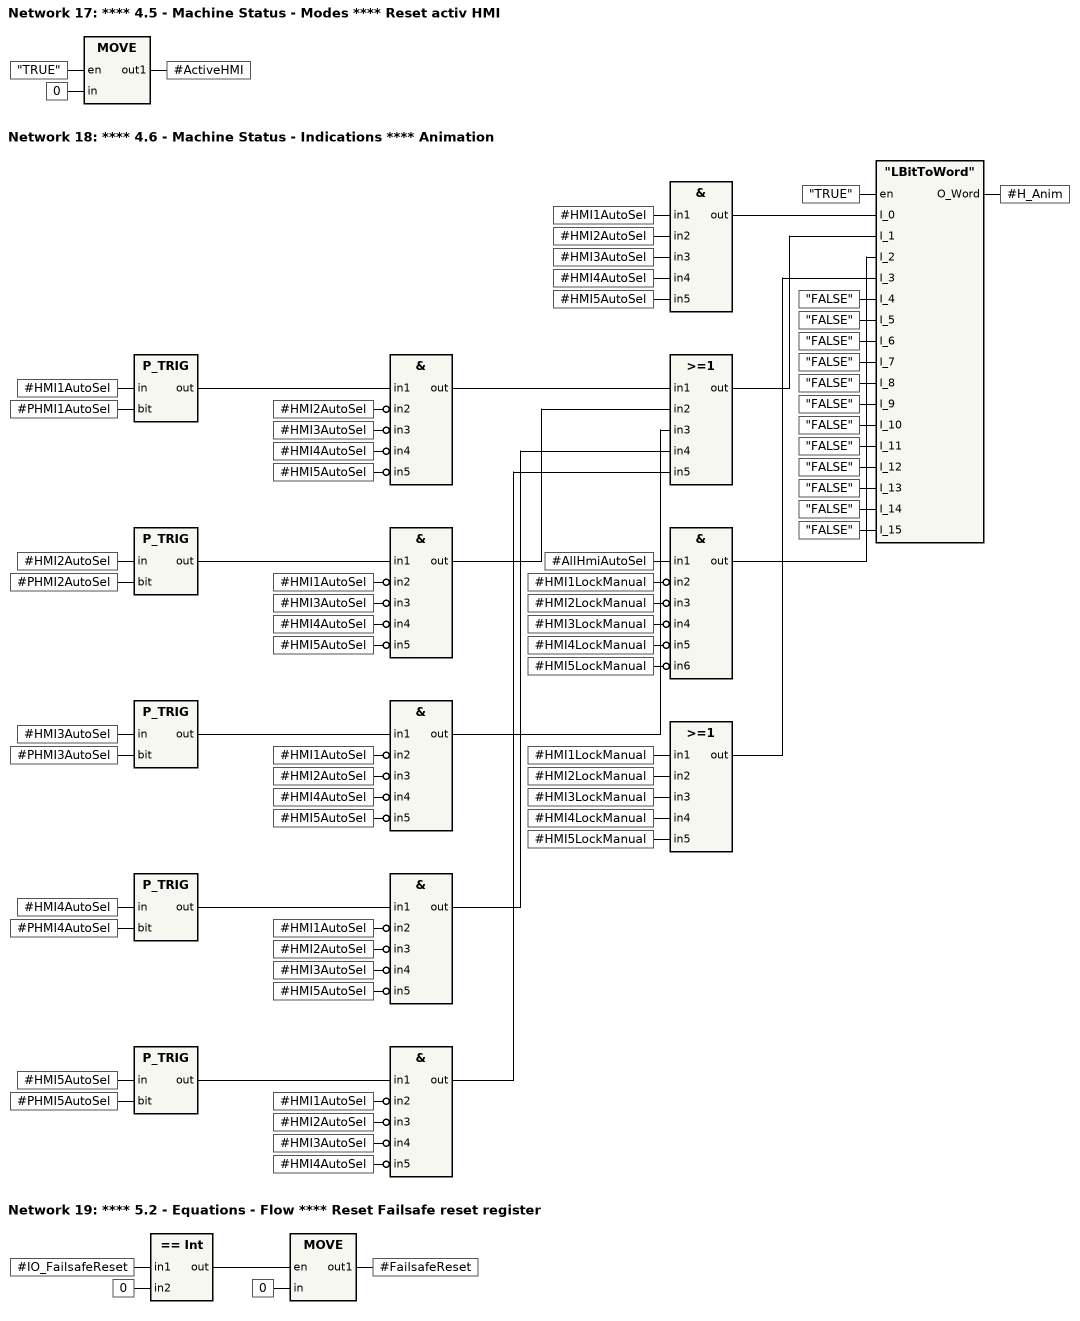
   IF "TRUE" THEN #ActiveHMI := 0; END_IF;
END_REGION

REGION Network 18: **** 4.6 - Machine Status - Indications **** Animation
   // Animation
   #_w1 := #HMI1AutoSel AND NOT #PHMI1AutoSel;   // rising edge
   #PHMI1AutoSel := #HMI1AutoSel;
   #_w2 := #HMI2AutoSel AND NOT #PHMI2AutoSel;   // rising edge
   #PHMI2AutoSel := #HMI2AutoSel;
   #_w3 := #HMI3AutoSel AND NOT #PHMI3AutoSel;   // rising edge
   #PHMI3AutoSel := #HMI3AutoSel;
   #_w4 := #HMI4AutoSel AND NOT #PHMI4AutoSel;   // rising edge
   #PHMI4AutoSel := #HMI4AutoSel;
   #_w5 := #HMI5AutoSel AND NOT #PHMI5AutoSel;   // rising edge
   #PHMI5AutoSel := #HMI5AutoSel;
   IF "TRUE" THEN
       "LBitToWord"(I_0 := #HMI1AutoSel AND #HMI2AutoSel AND #HMI3AutoSel AND #HMI4AutoSel AND #HMI5AutoSel,
                    I_1 := (#_w1 AND NOT #HMI2AutoSel AND NOT #HMI3AutoSel AND NOT #HMI4AutoSel AND NOT #HMI5AutoSel) OR (#_w2 AND NOT #HMI1AutoSel AND NOT #HMI3AutoSel AND NOT #HMI4AutoSel AND NOT #HMI5AutoSel) OR (#_w3 AND NOT #HMI1AutoSel AND NOT #HMI2AutoSel AND NOT #HMI4AutoSel AND NOT #HMI5AutoSel) OR (#_w4 AND NOT #HMI1AutoSel AND NOT #HMI2AutoSel AND NOT #HMI3AutoSel AND NOT #HMI5AutoSel) OR (#_w5 AND NOT #HMI1AutoSel AND NOT #HMI2AutoSel AND NOT #HMI3AutoSel AND NOT #HMI4AutoSel),
                    I_2 := #AllHmiAutoSel AND NOT #HMI1LockManual AND NOT #HMI2LockManual AND NOT #HMI3LockManual AND NOT #HMI4LockManual AND NOT #HMI5LockManual,
                    I_3 := #HMI1LockManual OR #HMI2LockManual OR #HMI3LockManual OR #HMI4LockManual OR #HMI5LockManual,
                    I_4 := "FALSE",
                    I_5 := "FALSE",
                    I_6 := "FALSE",
                    I_7 := "FALSE",
                    I_8 := "FALSE",
                    I_9 := "FALSE",
                    I_10 := "FALSE",
                    I_11 := "FALSE",
                    I_12 := "FALSE",
                    I_13 := "FALSE",
                    I_14 := "FALSE",
                    I_15 := "FALSE",
                    O_Word => #H_Anim);
   END_IF;
END_REGION

REGION Network 19: **** 5.2 - Equations - Flow **** Reset Failsafe reset register
   // Reset Failsafe reset register
   IF #IO_FailsafeReset = 0 THEN #FailsafeReset := 0; END_IF;
END_REGION

REGION Network 20: **** 5.2 - Equations - Flow **** Move 6 to the failsafe register when Alarm reset is slected on the HMI
   // Move 6 to the failsafe register when Alarm reset is slected on the HMI
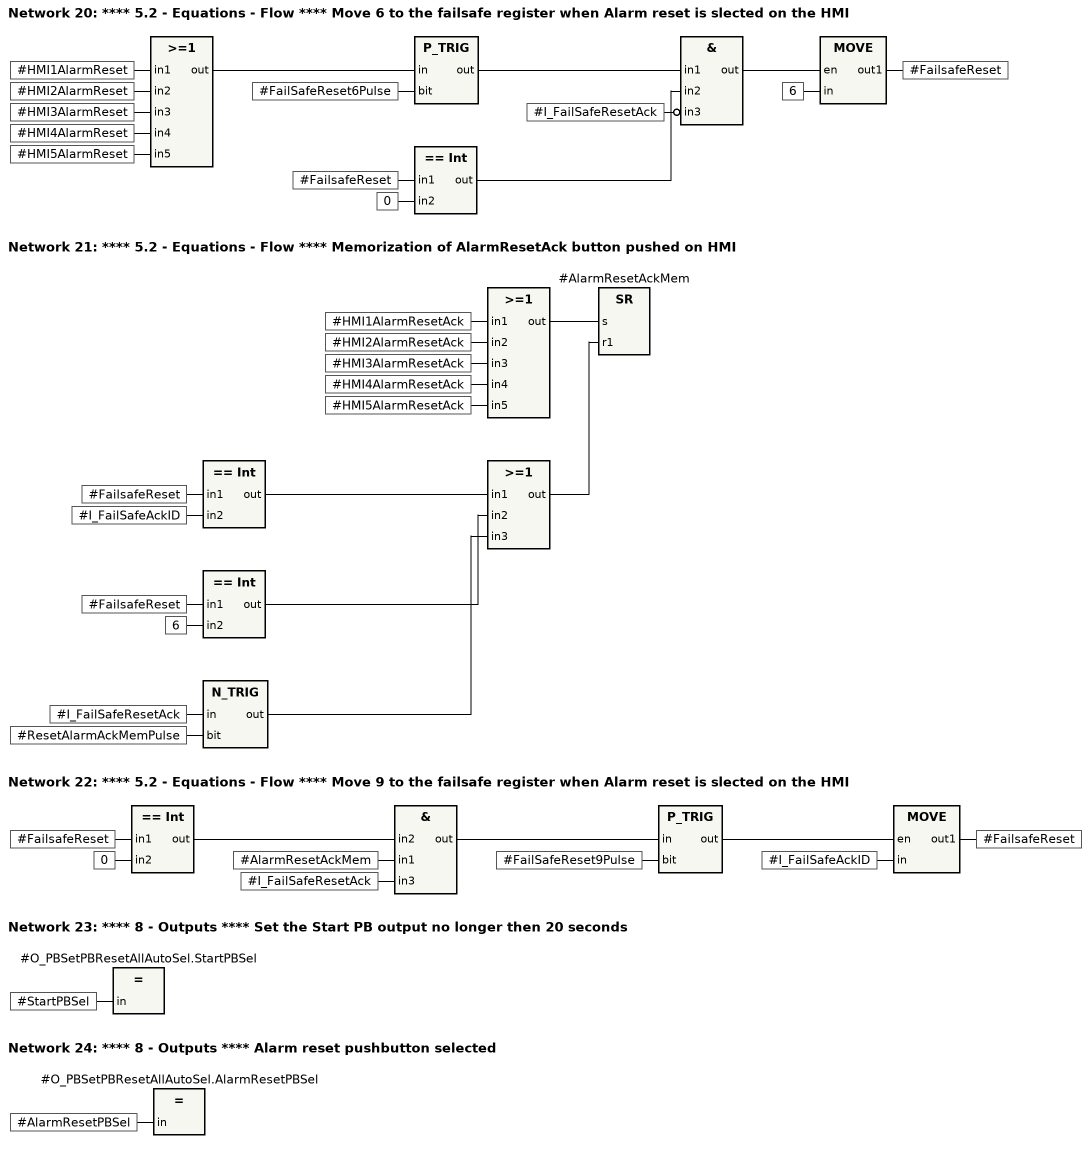
   #_w1 := #HMI1AlarmReset OR #HMI2AlarmReset OR #HMI3AlarmReset OR #HMI4AlarmReset OR #HMI5AlarmReset;
   #_w2 := #_w1 AND NOT #FailSafeReset6Pulse;   // rising edge
   #FailSafeReset6Pulse := #_w1;
   IF #_w2 AND (#FailsafeReset = 0) AND NOT #I_FailSafeResetAck THEN #FailsafeReset := 6; END_IF;
END_REGION

REGION Network 21: **** 5.2 - Equations - Flow **** Memorization of AlarmResetAck button pushed on HMI
   // Memorization of AlarmResetAck button pushed on HMI
   #_w1 := NOT #I_FailSafeResetAck AND #ResetAlarmAckMemPulse;   // falling edge
   #ResetAlarmAckMemPulse := #I_FailSafeResetAck;
   IF #HMI1AlarmResetAck OR #HMI2AlarmResetAck OR #HMI3AlarmResetAck OR #HMI4AlarmResetAck OR #HMI5AlarmResetAck THEN
       #AlarmResetAckMem := TRUE;   // SR flip-flop
   END_IF;
   IF (#FailsafeReset = #I_FailSafeAckID) OR (#FailsafeReset = 6) OR #_w1 THEN
       #AlarmResetAckMem := FALSE;
   END_IF;
END_REGION

REGION Network 22: **** 5.2 - Equations - Flow **** Move 9 to the failsafe register when Alarm reset is slected on the HMI
   // Move 9 to the failsafe register when Alarm reset is slected on the HMI
   #_w1 := (#FailsafeReset = 0) AND #AlarmResetAckMem AND #I_FailSafeResetAck;
   #_w2 := #_w1 AND NOT #FailSafeReset9Pulse;   // rising edge
   #FailSafeReset9Pulse := #_w1;
   IF #_w2 THEN #FailsafeReset := #I_FailSafeAckID; END_IF;
END_REGION

REGION Network 23: **** 8 - Outputs **** Set the Start PB output no longer then 20 seconds
   // Set the Start PB output no longer then 20 seconds
   #O_PBSetPBResetAllAutoSel.StartPBSel := #StartPBSel;
END_REGION

REGION Network 24: **** 8 - Outputs **** Alarm reset pushbutton selected
   // Alarm reset pushbutton selected
   #O_PBSetPBResetAllAutoSel.AlarmResetPBSel := #AlarmResetPBSel;
END_REGION

REGION Network 25: **** 8 - Outputs **** Set PB activated
   // Set PB activated
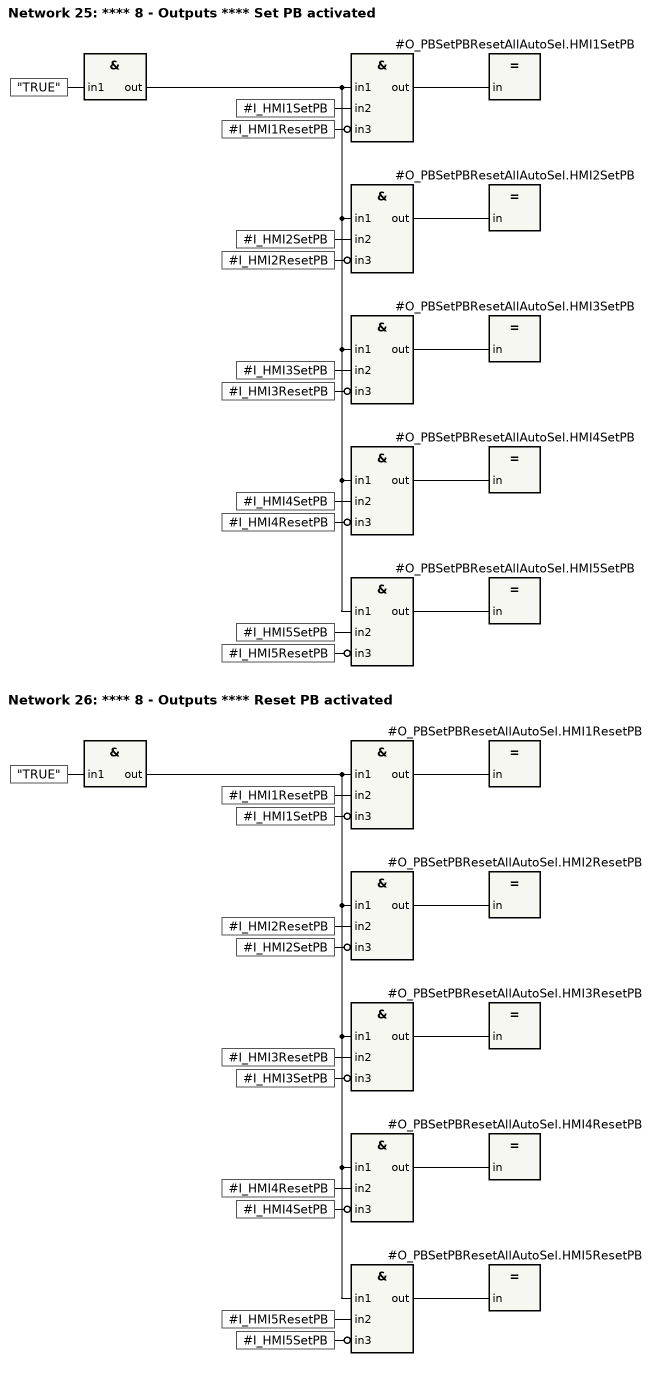
   #O_PBSetPBResetAllAutoSel.HMI1SetPB := "TRUE" AND #I_HMI1SetPB AND NOT #I_HMI1ResetPB;
   #O_PBSetPBResetAllAutoSel.HMI2SetPB := "TRUE" AND #I_HMI2SetPB AND NOT #I_HMI2ResetPB;
   #O_PBSetPBResetAllAutoSel.HMI3SetPB := "TRUE" AND #I_HMI3SetPB AND NOT #I_HMI3ResetPB;
   #O_PBSetPBResetAllAutoSel.HMI4SetPB := "TRUE" AND #I_HMI4SetPB AND NOT #I_HMI4ResetPB;
   #O_PBSetPBResetAllAutoSel.HMI5SetPB := "TRUE" AND #I_HMI5SetPB AND NOT #I_HMI5ResetPB;
END_REGION

REGION Network 26: **** 8 - Outputs **** Reset PB activated
   // Reset PB activated
   #O_PBSetPBResetAllAutoSel.HMI1ResetPB := "TRUE" AND #I_HMI1ResetPB AND NOT #I_HMI1SetPB;
   #O_PBSetPBResetAllAutoSel.HMI2ResetPB := "TRUE" AND #I_HMI2ResetPB AND NOT #I_HMI2SetPB;
   #O_PBSetPBResetAllAutoSel.HMI3ResetPB := "TRUE" AND #I_HMI3ResetPB AND NOT #I_HMI3SetPB;
   #O_PBSetPBResetAllAutoSel.HMI4ResetPB := "TRUE" AND #I_HMI4ResetPB AND NOT #I_HMI4SetPB;
   #O_PBSetPBResetAllAutoSel.HMI5ResetPB := "TRUE" AND #I_HMI5ResetPB AND NOT #I_HMI5SetPB;
END_REGION

REGION Network 27: **** 8 - Outputs **** All HMI Auto Sel
   // All HMI Auto Sel
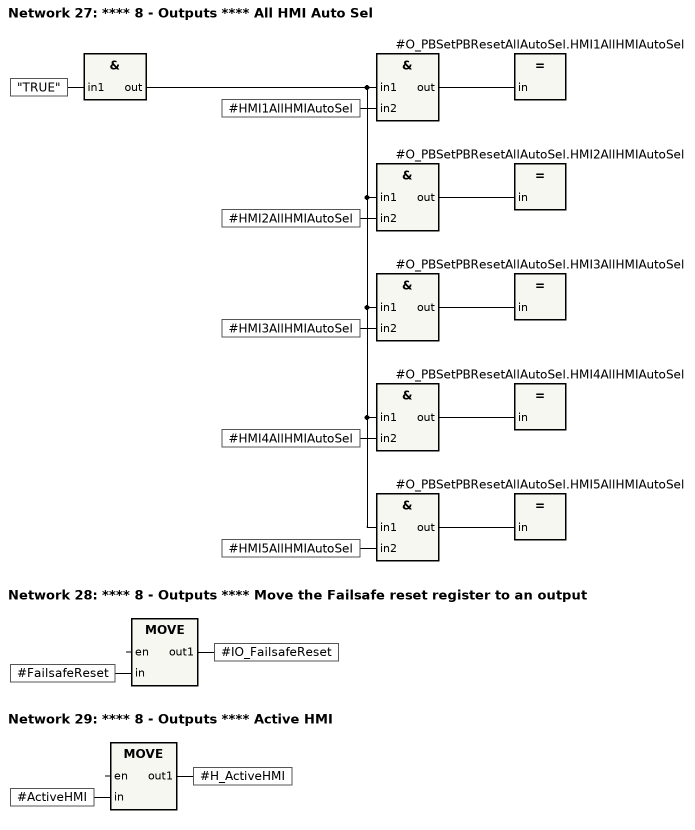
   #O_PBSetPBResetAllAutoSel.HMI1AllHMIAutoSel := "TRUE" AND #HMI1AllHMIAutoSel;
   #O_PBSetPBResetAllAutoSel.HMI2AllHMIAutoSel := "TRUE" AND #HMI2AllHMIAutoSel;
   #O_PBSetPBResetAllAutoSel.HMI3AllHMIAutoSel := "TRUE" AND #HMI3AllHMIAutoSel;
   #O_PBSetPBResetAllAutoSel.HMI4AllHMIAutoSel := "TRUE" AND #HMI4AllHMIAutoSel;
   #O_PBSetPBResetAllAutoSel.HMI5AllHMIAutoSel := "TRUE" AND #HMI5AllHMIAutoSel;
END_REGION

REGION Network 28: **** 8 - Outputs **** Move the Failsafe reset register to an output
   // Move the Failsafe reset register to an output
   #IO_FailsafeReset := #FailsafeReset;
END_REGION

REGION Network 29: **** 8 - Outputs **** Active HMI
   // Active HMI
   #H_ActiveHMI := #ActiveHMI;
END_REGION
END_FUNCTION_BLOCK
